DATA_BLOCK "IOManger.Output"
TITLE =
AUTHOR : EA
FAMILY : SIM
NAME : Inputs
VERSION : 0.1


  STRUCT
   in : ARRAY  [0 .. 512 ] OF BYTE ;
  END_STRUCT ;
BEGIN
   in[0] := B#16#0;
   in[1] := B#16#0;
   in[2] := B#16#0;
   in[3] := B#16#0;
   in[4] := B#16#0;
   in[5] := B#16#0;
   in[6] := B#16#0;
   in[7] := B#16#0;
   in[8] := B#16#0;
   in[9] := B#16#0;
   in[10] := B#16#0;
   in[11] := B#16#0;
   in[12] := B#16#0;
   in[13] := B#16#0;
   in[14] := B#16#0;
   in[15] := B#16#0;
   in[16] := B#16#0;
   in[17] := B#16#0;
   in[18] := B#16#0;
   in[19] := B#16#0;
   in[20] := B#16#0;
   in[21] := B#16#0;
   in[22] := B#16#0;
   in[23] := B#16#0;
   in[24] := B#16#0;
   in[25] := B#16#0;
   in[26] := B#16#0;
   in[27] := B#16#0;
   in[28] := B#16#0;
   in[29] := B#16#0;
   in[30] := B#16#0;
   in[31] := B#16#0;
   in[32] := B#16#0;
   in[33] := B#16#0;
   in[34] := B#16#0;
   in[35] := B#16#0;
   in[36] := B#16#0;
   in[37] := B#16#0;
   in[38] := B#16#0;
   in[39] := B#16#0;
   in[40] := B#16#0;
   in[41] := B#16#0;
   in[42] := B#16#0;
   in[43] := B#16#0;
   in[44] := B#16#0;
   in[45] := B#16#0;
   in[46] := B#16#0;
   in[47] := B#16#0;
   in[48] := B#16#0;
   in[49] := B#16#0;
   in[50] := B#16#0;
   in[51] := B#16#0;
   in[52] := B#16#0;
   in[53] := B#16#0;
   in[54] := B#16#0;
   in[55] := B#16#0;
   in[56] := B#16#0;
   in[57] := B#16#0;
   in[58] := B#16#0;
   in[59] := B#16#0;
   in[60] := B#16#0;
   in[61] := B#16#0;
   in[62] := B#16#0;
   in[63] := B#16#0;
   in[64] := B#16#0;
   in[65] := B#16#0;
   in[66] := B#16#0;
   in[67] := B#16#0;
   in[68] := B#16#0;
   in[69] := B#16#0;
   in[70] := B#16#0;
   in[71] := B#16#0;
   in[72] := B#16#0;
   in[73] := B#16#0;
   in[74] := B#16#0;
   in[75] := B#16#0;
   in[76] := B#16#0;
   in[77] := B#16#0;
   in[78] := B#16#0;
   in[79] := B#16#0;
   in[80] := B#16#0;
   in[81] := B#16#0;
   in[82] := B#16#0;
   in[83] := B#16#0;
   in[84] := B#16#0;
   in[85] := B#16#0;
   in[86] := B#16#0;
   in[87] := B#16#0;
   in[88] := B#16#0;
   in[89] := B#16#0;
   in[90] := B#16#0;
   in[91] := B#16#0;
   in[92] := B#16#0;
   in[93] := B#16#0;
   in[94] := B#16#0;
   in[95] := B#16#0;
   in[96] := B#16#0;
   in[97] := B#16#0;
   in[98] := B#16#0;
   in[99] := B#16#0;
   in[100] := B#16#0;
   in[101] := B#16#0;
   in[102] := B#16#0;
   in[103] := B#16#0;
   in[104] := B#16#0;
   in[105] := B#16#0;
   in[106] := B#16#0;
   in[107] := B#16#0;
   in[108] := B#16#0;
   in[109] := B#16#0;
   in[110] := B#16#0;
   in[111] := B#16#0;
   in[112] := B#16#0;
   in[113] := B#16#0;
   in[114] := B#16#0;
   in[115] := B#16#0;
   in[116] := B#16#0;
   in[117] := B#16#0;
   in[118] := B#16#0;
   in[119] := B#16#0;
   in[120] := B#16#0;
   in[121] := B#16#0;
   in[122] := B#16#0;
   in[123] := B#16#0;
   in[124] := B#16#0;
   in[125] := B#16#0;
   in[126] := B#16#0;
   in[127] := B#16#0;
   in[128] := B#16#0;
   in[129] := B#16#0;
   in[130] := B#16#0;
   in[131] := B#16#0;
   in[132] := B#16#0;
   in[133] := B#16#0;
   in[134] := B#16#0;
   in[135] := B#16#0;
   in[136] := B#16#0;
   in[137] := B#16#0;
   in[138] := B#16#0;
   in[139] := B#16#0;
   in[140] := B#16#0;
   in[141] := B#16#0;
   in[142] := B#16#0;
   in[143] := B#16#0;
   in[144] := B#16#0;
   in[145] := B#16#0;
   in[146] := B#16#0;
   in[147] := B#16#0;
   in[148] := B#16#0;
   in[149] := B#16#0;
   in[150] := B#16#0;
   in[151] := B#16#0;
   in[152] := B#16#0;
   in[153] := B#16#0;
   in[154] := B#16#0;
   in[155] := B#16#0;
   in[156] := B#16#0;
   in[157] := B#16#0;
   in[158] := B#16#0;
   in[159] := B#16#0;
   in[160] := B#16#0;
   in[161] := B#16#0;
   in[162] := B#16#0;
   in[163] := B#16#0;
   in[164] := B#16#0;
   in[165] := B#16#0;
   in[166] := B#16#0;
   in[167] := B#16#0;
   in[168] := B#16#0;
   in[169] := B#16#0;
   in[170] := B#16#0;
   in[171] := B#16#0;
   in[172] := B#16#0;
   in[173] := B#16#0;
   in[174] := B#16#0;
   in[175] := B#16#0;
   in[176] := B#16#0;
   in[177] := B#16#0;
   in[178] := B#16#0;
   in[179] := B#16#0;
   in[180] := B#16#0;
   in[181] := B#16#0;
   in[182] := B#16#0;
   in[183] := B#16#0;
   in[184] := B#16#0;
   in[185] := B#16#0;
   in[186] := B#16#0;
   in[187] := B#16#0;
   in[188] := B#16#0;
   in[189] := B#16#0;
   in[190] := B#16#0;
   in[191] := B#16#0;
   in[192] := B#16#0;
   in[193] := B#16#0;
   in[194] := B#16#0;
   in[195] := B#16#0;
   in[196] := B#16#0;
   in[197] := B#16#0;
   in[198] := B#16#0;
   in[199] := B#16#0;
   in[200] := B#16#0;
   in[201] := B#16#0;
   in[202] := B#16#0;
   in[203] := B#16#0;
   in[204] := B#16#0;
   in[205] := B#16#0;
   in[206] := B#16#0;
   in[207] := B#16#0;
   in[208] := B#16#0;
   in[209] := B#16#0;
   in[210] := B#16#0;
   in[211] := B#16#0;
   in[212] := B#16#0;
   in[213] := B#16#0;
   in[214] := B#16#0;
   in[215] := B#16#0;
   in[216] := B#16#0;
   in[217] := B#16#0;
   in[218] := B#16#0;
   in[219] := B#16#0;
   in[220] := B#16#0;
   in[221] := B#16#0;
   in[222] := B#16#0;
   in[223] := B#16#0;
   in[224] := B#16#0;
   in[225] := B#16#0;
   in[226] := B#16#0;
   in[227] := B#16#0;
   in[228] := B#16#0;
   in[229] := B#16#0;
   in[230] := B#16#0;
   in[231] := B#16#0;
   in[232] := B#16#0;
   in[233] := B#16#0;
   in[234] := B#16#0;
   in[235] := B#16#0;
   in[236] := B#16#0;
   in[237] := B#16#0;
   in[238] := B#16#0;
   in[239] := B#16#0;
   in[240] := B#16#0;
   in[241] := B#16#0;
   in[242] := B#16#0;
   in[243] := B#16#0;
   in[244] := B#16#0;
   in[245] := B#16#0;
   in[246] := B#16#0;
   in[247] := B#16#0;
   in[248] := B#16#0;
   in[249] := B#16#0;
   in[250] := B#16#0;
   in[251] := B#16#0;
   in[252] := B#16#0;
   in[253] := B#16#0;
   in[254] := B#16#0;
   in[255] := B#16#0;
   in[256] := B#16#0;
   in[257] := B#16#0;
   in[258] := B#16#0;
   in[259] := B#16#0;
   in[260] := B#16#0;
   in[261] := B#16#0;
   in[262] := B#16#0;
   in[263] := B#16#0;
   in[264] := B#16#0;
   in[265] := B#16#0;
   in[266] := B#16#0;
   in[267] := B#16#0;
   in[268] := B#16#0;
   in[269] := B#16#0;
   in[270] := B#16#0;
   in[271] := B#16#0;
   in[272] := B#16#0;
   in[273] := B#16#0;
   in[274] := B#16#0;
   in[275] := B#16#0;
   in[276] := B#16#0;
   in[277] := B#16#0;
   in[278] := B#16#0;
   in[279] := B#16#0;
   in[280] := B#16#0;
   in[281] := B#16#0;
   in[282] := B#16#0;
   in[283] := B#16#0;
   in[284] := B#16#0;
   in[285] := B#16#0;
   in[286] := B#16#0;
   in[287] := B#16#0;
   in[288] := B#16#0;
   in[289] := B#16#0;
   in[290] := B#16#0;
   in[291] := B#16#0;
   in[292] := B#16#0;
   in[293] := B#16#0;
   in[294] := B#16#0;
   in[295] := B#16#0;
   in[296] := B#16#0;
   in[297] := B#16#0;
   in[298] := B#16#0;
   in[299] := B#16#0;
   in[300] := B#16#0;
   in[301] := B#16#0;
   in[302] := B#16#0;
   in[303] := B#16#0;
   in[304] := B#16#0;
   in[305] := B#16#0;
   in[306] := B#16#0;
   in[307] := B#16#0;
   in[308] := B#16#0;
   in[309] := B#16#0;
   in[310] := B#16#0;
   in[311] := B#16#0;
   in[312] := B#16#0;
   in[313] := B#16#0;
   in[314] := B#16#0;
   in[315] := B#16#0;
   in[316] := B#16#0;
   in[317] := B#16#0;
   in[318] := B#16#0;
   in[319] := B#16#0;
   in[320] := B#16#0;
   in[321] := B#16#0;
   in[322] := B#16#0;
   in[323] := B#16#0;
   in[324] := B#16#0;
   in[325] := B#16#0;
   in[326] := B#16#0;
   in[327] := B#16#0;
   in[328] := B#16#0;
   in[329] := B#16#0;
   in[330] := B#16#0;
   in[331] := B#16#0;
   in[332] := B#16#0;
   in[333] := B#16#0;
   in[334] := B#16#0;
   in[335] := B#16#0;
   in[336] := B#16#0;
   in[337] := B#16#0;
   in[338] := B#16#0;
   in[339] := B#16#0;
   in[340] := B#16#0;
   in[341] := B#16#0;
   in[342] := B#16#0;
   in[343] := B#16#0;
   in[344] := B#16#0;
   in[345] := B#16#0;
   in[346] := B#16#0;
   in[347] := B#16#0;
   in[348] := B#16#0;
   in[349] := B#16#0;
   in[350] := B#16#0;
   in[351] := B#16#0;
   in[352] := B#16#0;
   in[353] := B#16#0;
   in[354] := B#16#0;
   in[355] := B#16#0;
   in[356] := B#16#0;
   in[357] := B#16#0;
   in[358] := B#16#0;
   in[359] := B#16#0;
   in[360] := B#16#0;
   in[361] := B#16#0;
   in[362] := B#16#0;
   in[363] := B#16#0;
   in[364] := B#16#0;
   in[365] := B#16#0;
   in[366] := B#16#0;
   in[367] := B#16#0;
   in[368] := B#16#0;
   in[369] := B#16#0;
   in[370] := B#16#0;
   in[371] := B#16#0;
   in[372] := B#16#0;
   in[373] := B#16#0;
   in[374] := B#16#0;
   in[375] := B#16#0;
   in[376] := B#16#0;
   in[377] := B#16#0;
   in[378] := B#16#0;
   in[379] := B#16#0;
   in[380] := B#16#0;
   in[381] := B#16#0;
   in[382] := B#16#0;
   in[383] := B#16#0;
   in[384] := B#16#0;
   in[385] := B#16#0;
   in[386] := B#16#0;
   in[387] := B#16#0;
   in[388] := B#16#0;
   in[389] := B#16#0;
   in[390] := B#16#0;
   in[391] := B#16#0;
   in[392] := B#16#0;
   in[393] := B#16#0;
   in[394] := B#16#0;
   in[395] := B#16#0;
   in[396] := B#16#0;
   in[397] := B#16#0;
   in[398] := B#16#0;
   in[399] := B#16#0;
   in[400] := B#16#0;
   in[401] := B#16#0;
   in[402] := B#16#0;
   in[403] := B#16#0;
   in[404] := B#16#0;
   in[405] := B#16#0;
   in[406] := B#16#0;
   in[407] := B#16#0;
   in[408] := B#16#0;
   in[409] := B#16#0;
   in[410] := B#16#0;
   in[411] := B#16#0;
   in[412] := B#16#0;
   in[413] := B#16#0;
   in[414] := B#16#0;
   in[415] := B#16#0;
   in[416] := B#16#0;
   in[417] := B#16#0;
   in[418] := B#16#0;
   in[419] := B#16#0;
   in[420] := B#16#0;
   in[421] := B#16#0;
   in[422] := B#16#0;
   in[423] := B#16#0;
   in[424] := B#16#0;
   in[425] := B#16#0;
   in[426] := B#16#0;
   in[427] := B#16#0;
   in[428] := B#16#0;
   in[429] := B#16#0;
   in[430] := B#16#0;
   in[431] := B#16#0;
   in[432] := B#16#0;
   in[433] := B#16#0;
   in[434] := B#16#0;
   in[435] := B#16#0;
   in[436] := B#16#0;
   in[437] := B#16#0;
   in[438] := B#16#0;
   in[439] := B#16#0;
   in[440] := B#16#0;
   in[441] := B#16#0;
   in[442] := B#16#0;
   in[443] := B#16#0;
   in[444] := B#16#0;
   in[445] := B#16#0;
   in[446] := B#16#0;
   in[447] := B#16#0;
   in[448] := B#16#0;
   in[449] := B#16#0;
   in[450] := B#16#0;
   in[451] := B#16#0;
   in[452] := B#16#0;
   in[453] := B#16#0;
   in[454] := B#16#0;
   in[455] := B#16#0;
   in[456] := B#16#0;
   in[457] := B#16#0;
   in[458] := B#16#0;
   in[459] := B#16#0;
   in[460] := B#16#0;
   in[461] := B#16#0;
   in[462] := B#16#0;
   in[463] := B#16#0;
   in[464] := B#16#0;
   in[465] := B#16#0;
   in[466] := B#16#0;
   in[467] := B#16#0;
   in[468] := B#16#0;
   in[469] := B#16#0;
   in[470] := B#16#0;
   in[471] := B#16#0;
   in[472] := B#16#0;
   in[473] := B#16#0;
   in[474] := B#16#0;
   in[475] := B#16#0;
   in[476] := B#16#0;
   in[477] := B#16#0;
   in[478] := B#16#0;
   in[479] := B#16#0;
   in[480] := B#16#0;
   in[481] := B#16#0;
   in[482] := B#16#0;
   in[483] := B#16#0;
   in[484] := B#16#0;
   in[485] := B#16#0;
   in[486] := B#16#0;
   in[487] := B#16#0;
   in[488] := B#16#0;
   in[489] := B#16#0;
   in[490] := B#16#0;
   in[491] := B#16#0;
   in[492] := B#16#0;
   in[493] := B#16#0;
   in[494] := B#16#0;
   in[495] := B#16#0;
   in[496] := B#16#0;
   in[497] := B#16#0;
   in[498] := B#16#0;
   in[499] := B#16#0;
   in[500] := B#16#0;
   in[501] := B#16#0;
   in[502] := B#16#0;
   in[503] := B#16#0;
   in[504] := B#16#0;
   in[505] := B#16#0;
   in[506] := B#16#0;
   in[507] := B#16#0;
   in[508] := B#16#0;
   in[509] := B#16#0;
   in[510] := B#16#0;
   in[511] := B#16#0;
   in[512] := B#16#0;
END_DATA_BLOCK

